DATA_BLOCK "DB_BatchLog"
{ S7_Optimized_Access := 'TRUE' }
VERSION : 0.1
NON_RETAIN
   VAR
      WriteIndex : Int;
      TotalCount : DInt;
      Records { S7_SetPoint := 'False'} : Array[1..20] of "UDT_BatchRecord";
   END_VAR


BEGIN
   WriteIndex := 1;

END_DATA_BLOCK

